{attribute 'call_after_init'}
FUNCTION_BLOCK FB_evRangeCalculator_Test EXTENDS FB_TestSuite
VAR_INPUT
END_VAR
VAR_OUTPUT
END_VAR
VAR
END_VAR

BasicFunction();

METHOD BasicFunction
VAR_INPUT
END_VAR
VAR
    LastWord : WORD := 2#0000_0000_0000_0010;
END_VAR
TEST('CheckRanges');
//Upper limit equal
AssertTrue(
    F_eVRangeCalculator(300, 0) = 2#0000_0000_0000_0110,
    'Upper limit not inclusive');
//Lower limit equal
AssertTrue(
    F_eVRangeCalculator(300, 0) = 2#0000_0000_0000_0110,
    'Upper limit not inclusive');
//Mid range
AssertTrue(
    F_eVRangeCalculator(251, 0) = 2#0000_0000_0000_0010,
    'In range failed, whatever you did, it broke this really bad.');
//Out of range
AssertFalse(
    F_eVRangeCalculator(300.1, 0) = 2#0000_0000_0000_0010,
    'Out of range failed, whatever you did, it broke this really bad.');

TEST_FINISHED();

TEST('Negative eV failsafes');
//Negative eV
AssertTrue(
    F_eVRangeCalculator(-300, 0) = 16#FFFF,
    'Working with antimatter? Negative eV should failsafe to FFFF.');    

TEST_FINISHED();

TEST('Check hyst keeps');

AssertTrue(
    F_eVRangeCalculator(350, 2#0000_0000_0000_0010) = 2#0000_0000_0000_0110,
    'Moving up does not stick.');
    
AssertTrue(
    F_eVRangeCalculator(150, 2#0000_0000_0000_0010) = 2#0000_0000_0000_0011,
    'Moving down does not stick.');

TEST_FINISHED();

TEST('Check hyst drops');

AssertTrue(
    F_eVRangeCalculator(351, 2#0000_0000_0000_0010) = 2#0000_0000_0000_0100,
    'Moving up does not drop.');
    
AssertTrue(
    F_eVRangeCalculator(149, 2#0000_0000_0000_0010) = 2#0000_0000_0000_0001,
    'Moving down does not drop.');

TEST_FINISHED();

TEST_FINISHED_NAMED('FOO');
END_METHOD

END_FUNCTION_BLOCK

(* stored: Version 1.1.0.1, ProductVersion 3.1.4024.0
   POU FB_evRangeCalculator_Test: Id {e6bcc6ca-553c-488f-ba3b-eabce151236e}, SpecialFunc None
   Method BasicFunction: Id {2787ce06-fe9f-4a43-87a2-e050fc9f0a9f} *)
